{attribute addProperty BoxType "EL1254--0000"}
{attribute addProperty Id "ChannelAT %I*ARRAY[0..3] OF Channel_E4AEF59E3240ReservedEMPTY_STRUCTURE000LatchAT %I*Latch_BE22BB17544680WcStateAT %I*WcState_F855686C1620InfoDataAT %I*InfoData_7231B2DD80100"}
{attribute addProperty CRC "1780291789"}
{attribute addProperty SizeInBites "672"}
{attribute addProperty SizeInBytes "84"}
TYPE EL1254_D71D85A4 :
STRUCT
	{attribute addProperty Name "Channel"}
	Channel : ARRAY[0..3] OF Channel_E4AEF59E;
	{attribute addProperty Name "Reserved"}
	Reserved : EMPTY_STRUCTURE;
	{attribute addProperty Name "Latch"}
	Latch : Latch_BE22BB17;
	{attribute addProperty Name "WcState"}
	WcState : WcState_F855686C;
	{attribute addProperty Name "InfoData"}
	InfoData : InfoData_7231B2DD;
END_STRUCT
END_TYPE

(* stored: Version 1.2.0.0, ProductVersion 3.1.4024.9
   DUT EL1254_D71D85A4: Id {6810f849-c51d-4b37-b81d-2f47e214978f} *)
